// TIA Portal V17 export
// export: Created 2023-02-25T15:47:10.9232914Z, ExportSetting WithDefaults, DisplayName Totally Integrated Automation Portal, DisplayVersion V17, DisplayName TIA Portal Openness, DisplayVersion V17, DisplayName TIA Portal Version Control Interface, DisplayVersion V17, DisplayName TIA Portal Test Suite Advanced, DisplayVersion V17, DisplayName STEP 7 Professional, DisplayVersion V17, DisplayName SIMATIC Energy Suite, DisplayVersion V17, DisplayName STEP 7 Safety, DisplayVersion V17, DisplayName WinCC Professional, DisplayVersion V17
FUNCTION "LOG_ManualControle" : Void   // FC10, LAD
{ S7_Optimized_Access := 'TRUE' }
VERSION : 0.1
// stored: AutoNumber true, IsIECCheckEnabled false, SetENOAutomatically false, UDAEnableTagReadback false
   VAR_INPUT
      StartLine : Bool;
      StopLine : Bool;
      ModeManual : Bool;
      T1Button : Bool;
      T2Button : Bool;
      T3Button : Bool;
      T4Button : Bool;
      WButton : Bool;
      SendLeftButton : Bool;
      SendForwardButton : Bool;
      SendRightButton : Bool;
   END_VAR
   VAR_OUTPUT
      ConveyorsManual : "stt_Conveyor";
   END_VAR
BEGIN

REGION Network 1: Call: ManualModule - C1
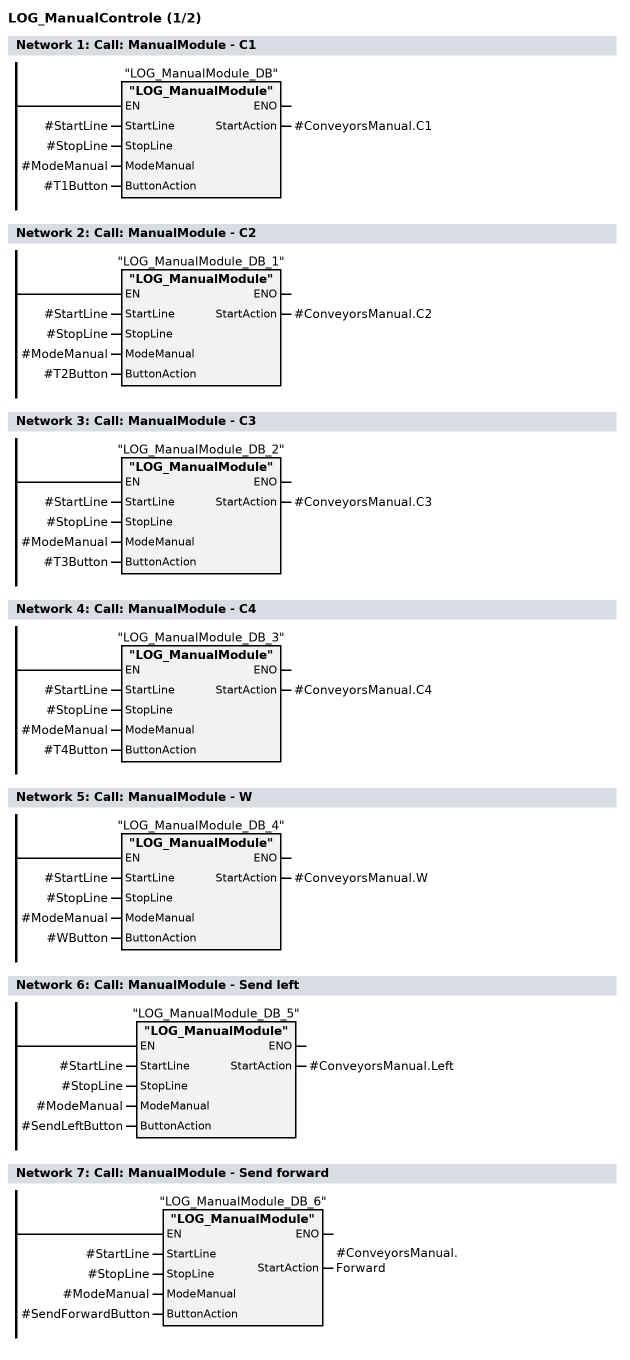
   RUNG wire#powerrail
      "LOG_ManualModule_DB"(StartLine := #StartLine, StopLine := #StopLine, ModeManual := #ModeManual, ButtonAction := #T1Button, StartAction => #ConveyorsManual.C1)
   END_RUNG
   // the same network as SCL:
   "LOG_ManualModule_DB"(StartLine := #StartLine,   // "LOG_ManualModule"
                         StopLine := #StopLine,
                         ModeManual := #ModeManual,
                         ButtonAction := #T1Button,
                         StartAction => #ConveyorsManual.C1);
END_REGION

REGION Network 2: Call: ManualModule - C2
   RUNG wire#powerrail
      "LOG_ManualModule_DB_1"(StartLine := #StartLine, StopLine := #StopLine, ModeManual := #ModeManual, ButtonAction := #T2Button, StartAction => #ConveyorsManual.C2)
   END_RUNG
   // the same network as SCL:
   "LOG_ManualModule_DB_1"(StartLine := #StartLine,   // "LOG_ManualModule"
                           StopLine := #StopLine,
                           ModeManual := #ModeManual,
                           ButtonAction := #T2Button,
                           StartAction => #ConveyorsManual.C2);
END_REGION

REGION Network 3: Call: ManualModule - C3
   RUNG wire#powerrail
      "LOG_ManualModule_DB_2"(StartLine := #StartLine, StopLine := #StopLine, ModeManual := #ModeManual, ButtonAction := #T3Button, StartAction => #ConveyorsManual.C3)
   END_RUNG
   // the same network as SCL:
   "LOG_ManualModule_DB_2"(StartLine := #StartLine,   // "LOG_ManualModule"
                           StopLine := #StopLine,
                           ModeManual := #ModeManual,
                           ButtonAction := #T3Button,
                           StartAction => #ConveyorsManual.C3);
END_REGION

REGION Network 4: Call: ManualModule - C4
   RUNG wire#powerrail
      "LOG_ManualModule_DB_3"(StartLine := #StartLine, StopLine := #StopLine, ModeManual := #ModeManual, ButtonAction := #T4Button, StartAction => #ConveyorsManual.C4)
   END_RUNG
   // the same network as SCL:
   "LOG_ManualModule_DB_3"(StartLine := #StartLine,   // "LOG_ManualModule"
                           StopLine := #StopLine,
                           ModeManual := #ModeManual,
                           ButtonAction := #T4Button,
                           StartAction => #ConveyorsManual.C4);
END_REGION

REGION Network 5: Call: ManualModule - W
   RUNG wire#powerrail
      "LOG_ManualModule_DB_4"(StartLine := #StartLine, StopLine := #StopLine, ModeManual := #ModeManual, ButtonAction := #WButton, StartAction => #ConveyorsManual.W)
   END_RUNG
   // the same network as SCL:
   "LOG_ManualModule_DB_4"(StartLine := #StartLine,   // "LOG_ManualModule"
                           StopLine := #StopLine,
                           ModeManual := #ModeManual,
                           ButtonAction := #WButton,
                           StartAction => #ConveyorsManual.W);
END_REGION

REGION Network 6: Call: ManualModule - Send left
   RUNG wire#powerrail
      "LOG_ManualModule_DB_5"(StartLine := #StartLine, StopLine := #StopLine, ModeManual := #ModeManual, ButtonAction := #SendLeftButton, StartAction => #ConveyorsManual.Left)
   END_RUNG
   // the same network as SCL:
   "LOG_ManualModule_DB_5"(StartLine := #StartLine,   // "LOG_ManualModule"
                           StopLine := #StopLine,
                           ModeManual := #ModeManual,
                           ButtonAction := #SendLeftButton,
                           StartAction => #ConveyorsManual.Left);
END_REGION

REGION Network 7: Call: ManualModule - Send forward
   RUNG wire#powerrail
      "LOG_ManualModule_DB_6"(StartLine := #StartLine, StopLine := #StopLine, ModeManual := #ModeManual, ButtonAction := #SendForwardButton, StartAction => #ConveyorsManual.Forward)
   END_RUNG
   // the same network as SCL:
   "LOG_ManualModule_DB_6"(StartLine := #StartLine,   // "LOG_ManualModule"
                           StopLine := #StopLine,
                           ModeManual := #ModeManual,
                           ButtonAction := #SendForwardButton,
                           StartAction => #ConveyorsManual.Forward);
END_REGION

REGION Network 8: Call: ManualModule - Send right
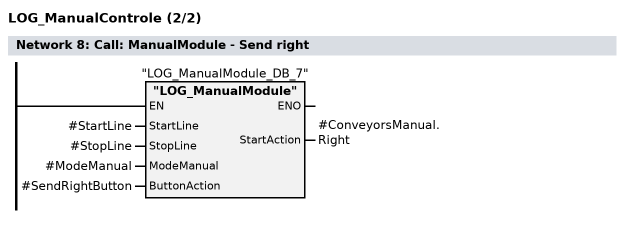
   RUNG wire#powerrail
      "LOG_ManualModule_DB_7"(StartLine := #StartLine, StopLine := #StopLine, ModeManual := #ModeManual, ButtonAction := #SendRightButton, StartAction => #ConveyorsManual.Right)
   END_RUNG
   // the same network as SCL:
   "LOG_ManualModule_DB_7"(StartLine := #StartLine,   // "LOG_ManualModule"
                           StopLine := #StopLine,
                           ModeManual := #ModeManual,
                           ButtonAction := #SendRightButton,
                           StartAction => #ConveyorsManual.Right);
END_REGION
END_FUNCTION
